FUNCTION_BLOCK LinearEncodedDrive_2Sensor EXTENDS FBA_LinearDrive IMPLEMENTS I_LinearEncodedDrive
VAR_INPUT
	drive : I_EncodedDrive;
	homeAt0 : BOOL;
	allowDualSideTraverse : BOOL; //allows motion between home to retractLimit
END_VAR
VAR_OUTPUT
	position : LREAL;
	velocity : LREAL;
END_VAR
VAR
	extendLimit AT %I* : BOOL;
	
	homePosition : LREAL;
	limitPosition : LREAL;
	
	calculation : (IDLE, EXTEND, RETRACT, CALCULATE, DONE);
END_VAR

override();

ready := bEnable AND NOT Active AND HomeSet;

PROPERTY Active : BOOL
GET
Active := drive.Active;
END_GET
END_PROPERTY

PROPERTY AtExtendLimit : BOOL
GET
AtExtendLimit := extendLimit <> sensorDefaultState;
END_GET
END_PROPERTY

METHOD PRIVATE calculatePositions : BOOL
(*
THIS METHOD IS ONLY TO BE CALLED IF homeAt0 IS FALSE

not all drives have their home sensor at the 0 position
the purpose of this method is to calculate the home position, under the assumption that the extend limit sensor is 0

implementation:
	start from home
	reach the extend limit and set position to 0
	return to the home sensor and set the home position to the current position
*)
CASE calculation OF
	IDLE:
		calculation := EXTEND;
		
	EXTEND:		
		IF AtExtendLimit THEN
			
			IF homeAt0 THEN
				limitPosition := CurrentPosition;
				calculation := RETRACT;
			
			ELSIF setPosition(newPosition := 0) THEN
				limitPosition := 0;
				calculation := RETRACT;
			END_IF
		
		ELSE
			moveContinuous(newDirection := MC_Negative_Direction);
		END_IF
		
	RETRACT:
		IF AtHome THEN
			
			IF homeAt0 THEN
				homePosition := 0;
				calculation := DONE;
			
			ELSE
				homePosition := CurrentPosition;
				calculation := DONE;
			END_IF
		
		ELSE
			moveContinuous(newDirection := MC_Positive_Direction);
		END_IF
		
	DONE:
		calculation := 0;
		calculatePositions := TRUE;
		
END_CASE
END_METHOD

PROPERTY CurrentPosition : LREAL
GET
CurrentPosition := position;
END_GET
END_PROPERTY

PROPERTY Error : BOOL
GET
error := drive.Error;
END_GET
END_PROPERTY

METHOD homingSequence : BOOL
(*
homing sequence is different for linear motion devices with limit sensors
*)
CASE step OF
	Homing.IDLE:
		reset();
		IF bEnable THEN
			step := Homing.START;
		END_IF
		
	Homing.START:
		IF AtHome THEN
			step := Homing.STOP;
			
		ELSIF AtExtendLimit THEN
			step := Homing.RETRY;
			
		ELSE
			moveContinuous(newDirection:= MC_Positive_Direction);
		END_IF
		
	Homing.STOP:
		IF stop() THEN
			step := Homing.DONE;
		END_IF
		
	Homing.DONE:
		homingComplete := TRUE;
		step := Homing.IDLE;
		
END_CASE
END_METHOD

METHOD moveAbsolute : BOOL
VAR_INPUT
	newTarget : LREAL;
END_VAR
(*
VAR_OUTPUT
	fault : BOOL;
END_VAR
*)
drive.moveAbsolute(newTarget:= newTarget);

moveAbsolute := drive.CurrentPosition = newTarget;
END_METHOD

METHOD moveContinuous : BOOL
VAR_INPUT
	//direction : BOOL; //direction (F = inwards, T = outwards)
	newDirection : MC_Direction;
END_VAR
drive.moveContinuous(newDirection:= newDirection);

direction := newDirection;
END_METHOD

METHOD moveRelative : BOOL
VAR_INPUT
	distance : LREAL;
END_VAR
drive.moveRelative(distance:= distance);
END_METHOD

METHOD PRIVATE override : BOOL
VAR_INPUT
END_VAR
(*
-at home and attempting to traverse outward
-at outer limit and attempting to traverse outward
-at inner limit and attempting to traverse inwards
*)
(*
inward = negative direction, negative velocity
outward = positive direction, positive velocity
*)

IF error THEN
	stop();
	reset();
	
ELSIF
	(AtHome AND (TargetPosition > CurrentPosition OR direction = MC_Positive_Direction)) OR
	(AtExtendLimit AND (TargetPosition > CurrentPosition OR direction = MC_Negative_Direction))
THEN
	stop();
END_IF
END_METHOD

METHOD reset : BOOL
VAR_INPUT
END_VAR
reset := drive.reset();
END_METHOD

METHOD setPosition : BOOL
VAR_INPUT
	newPosition : LREAL;
END_VAR
setPosition := drive.setPosition(newPosition:= newPosition);
END_METHOD

METHOD stop : BOOL
VAR_INPUT
END_VAR
drive.stop();
END_METHOD

PROPERTY TargetPosition : LREAL
GET
END_GET
END_PROPERTY

METHOD toHome : BOOL
VAR_INPUT
END_VAR
moveAbsolute(newTarget := homePosition);
END_METHOD

END_FUNCTION_BLOCK

(* stored: Version 1.1.0.1, ProductVersion 3.1.4024.11
   POU LinearEncodedDrive_2Sensor: Id {7c8236ed-0546-4a70-bd1c-508a9b819dac}, SpecialFunc None
   Folder Private: Id {fbf0c29e-ae6a-490d-b295-4aa7f22d20a1}
   Folder Properties: Id {22760fa6-a40f-4c6d-aa74-2480e3b707e0}
   Property Active: Id {9b3bc6dd-0e3f-4608-87c2-b8b44e8579bc}
   Get Get: Id {0ca1cd28-9432-42da-86f4-6139bbd45d2c}
   Property AtExtendLimit: Id {a2e60b92-cdee-42de-8b3f-315867de23ed}
   Get Get: Id {4545a776-2853-473c-9800-5c60f4e9846a}
   Method calculatePositions: Id {7affd250-9014-4192-91af-f8ea051feef0}
   Property CurrentPosition: Id {50bdea53-dbce-4047-a508-de920c329f34}
   Get Get: Id {bef4e104-c5b7-4454-aabc-d4fdc51e7ba9}
   Property Error: Id {38728739-ca79-442e-9eee-fe00c0f7c5e5}
   Get Get: Id {dbc122fe-0935-4b2d-bbd4-f7200feec772}
   Method homingSequence: Id {281986e6-28c9-4075-adab-180602cd765c}
   Method moveAbsolute: Id {4c6d4e38-d9c5-46ea-af0d-23af61edc0c8}
   Method moveContinuous: Id {009910ab-3cb6-4f78-a069-c011b0396d54}
   Method moveRelative: Id {17696c28-cd64-48d7-b362-d4d0b97ea37c}
   Method override: Id {b2d747e4-5c5c-4617-ae45-0343ceab3693}
   Method reset: Id {68478207-0aae-4f1a-b7a5-39fbcfcf99af}
   Method setPosition: Id {cf91cbdb-19e5-435f-a57e-c111bff59789}
   Method stop: Id {c3602783-d781-4e5d-a5b5-80a85037b469}
   Property TargetPosition: Id {82df4f12-cdac-43ea-94af-26d2c237b8a8}
   Get Get: Id {b4306c79-6a5b-4f2c-a157-5074dea5dd59}
   Method toHome: Id {02cc98d9-6d6b-4da0-b3ad-dd1be67ce24d} *)
